INTERFACE IEventLogger

METHOD Send : BOOL
VAR_INPUT
	eventType : Tc3_EventLogger.TcEventEntry;
	args : STRING(255);
END_VAR
END_METHOD

END_INTERFACE

(* stored: Version 1.1.0.1, ProductVersion 3.1.4024.11
   Itf IEventLogger: Id {1945e7b6-5c19-41b4-9662-b526d53fcdb6}
   Method Send: Id {88d52675-853f-42aa-b3d0-3dee57b05991} *)
